INTERFACE I_InterfaceBase EXTENDS __System.IQueryInterface

END_INTERFACE

(* stored: Version 1.1.0.1, ProductVersion 3.1.4024.12
   Itf I_InterfaceBase: Id {907487e3-14a0-4878-87d4-bc30e49de76c} *)
